TYPE Machine_typ :
STRUCT
	Cmd	: MachineCmd_typ;
	Sts	: MachineSts_typ;
END_STRUCT
END_TYPE

(* stored: Version 1.1.0.1, ProductVersion 3.1.4026.8
   DUT Machine_typ: Id {bab696e4-20d7-02e1-200d-c8d80adb2f41} *)
